FUNCTION_BLOCK FB_LamparaMemorizada_ST
// La lampara se enciende al accionar el pulsador de conexion
// La lampara se apaga al accionar el pulsador de desconexion
VAR
    Lampara AT %Q*: BOOL;
    PulsadorConexion AT %I*: BOOL;
    PulsadorDesconexion AT %I*: BOOL;
END_VAR

IF PulsadorDesconexion THEN
    Lampara := FALSE;
ELSIF PulsadorConexion THEN
    Lampara := TRUE;
END_IF;

END_FUNCTION_BLOCK

(* stored: Version 1.1.0.1, ProductVersion 3.1.4024.15
   POU FB_LamparaMemorizada_ST: Id {c5b457af-eab2-4eba-8e3c-68d932391f11}, SpecialFunc None *)
